(* PLC project Sin nombre, Desconocido Sin nombre 1 *)
(* stored: creationDateTime 2024-10-25T17:54:31, modificationDateTime 2024-10-26T15:27:06 *)

PROGRAM joystick
  VAR
    anguloBrazo AT %MW0.0 : INT := 0;  (* variable para guardar el angulo del brazo *)
  END_VAR
  VAR CONSTANT
    primerled AT %MW0.1 : INT := 40;  (* valor para comparar si hay mas de 45 grados *)
    segundoled AT %MW0.2 : INT := 90;  (* valor para comparar si hay mas de 90 grados *)
    tercerled AT %MW0.3 : INT := 120;  (* valor para comparar si hay mas de 120 grados *)
    cuartoled AT %MW0.4 : INT := 150;  (* valor para comparar si hay mas de 150 grados *)
  END_VAR
  VAR
    joystickEntrada AT %IW0.1 : INT;  (* lectura del sensor al mover la palanca a la derecha *)
  END_VAR
  VAR CONSTANT
    joystickDerecha AT %MW0.5 : INT := 1000;  (* valor para comparar si la palanca esta hacia la derecha *)
    joystickIzquierda AT %MW0.6 : INT := 10;  (* valor para comparar si la palanca esta hacia la izquierda *)
  END_VAR
  VAR
    led45grados AT %QX0.0 : BOOL := 0;  (* salida de led cuando hay mas de 45 grados *)
    led90grados AT %QX0.1 : BOOL := 0;  (* salida de led cuando hay mas de 90 grados *)
    led120grados AT %QX0.2 : BOOL := 0;  (* salida de led cuando hay mas de 120 grados *)
    led150grados AT %QX0.3 : BOOL := 0;  (* salida de led cuando hay mas de 150 grados *)
    relay AT %QX0.4 : BOOL := 0;  (* salida de relay que se activa con algun movimiento del joystick *)
  END_VAR
  VAR  (* added by the conversion: wires and edge detectors of the diagram *)
    _LE28_OUT : BOOL;
    _GE1_OUT : BOOL;
  END_VAR

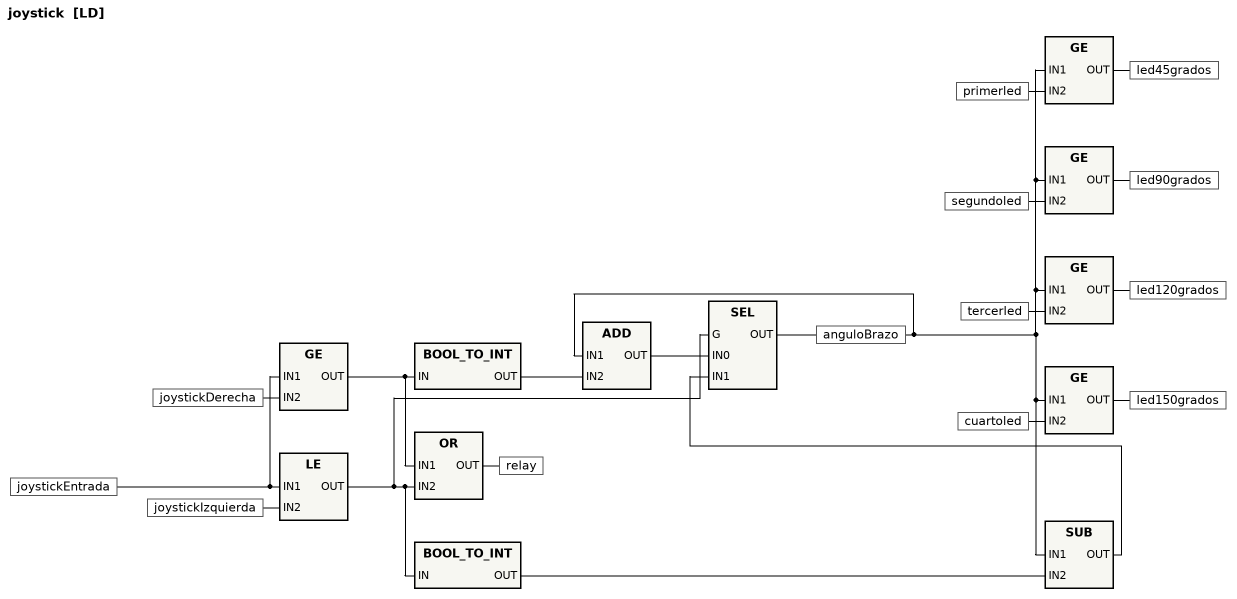
(* LD diagram, written out as Structured Text *)
led45grados := anguloBrazo >= primerled;
_LE28_OUT := joystickEntrada <= joystickIzquierda;
_GE1_OUT := joystickEntrada >= joystickDerecha;
anguloBrazo := SEL(_LE28_OUT, anguloBrazo + BOOL_TO_INT(_GE1_OUT), anguloBrazo - BOOL_TO_INT(_LE28_OUT));
led90grados := anguloBrazo >= segundoled;
led120grados := anguloBrazo >= tercerled;
led150grados := anguloBrazo >= cuartoled;
relay := _GE1_OUT OR _LE28_OUT;
END_PROGRAM

CONFIGURATION Config0
  RESOURCE Res0 ON PLC
    TASK task0(INTERVAL := T#20ms, PRIORITY := 0);
    PROGRAM instance0 WITH task0 : joystick;
  END_RESOURCE
END_CONFIGURATION
